TYPE U_UNION1 :
UNION
	aLights :		ARRAY[0..7] OF S_LIGHTS;
	aBits  : ARRAY[1..2] OF ST_Bits;
END_UNION
END_TYPE

(* stored: Version 1.1.0.1, ProductVersion 3.1.4024.10
   DUT U_UNION1: Id {d1a28e9f-3886-45c8-af49-e0c1694fe202} *)
